LIN {X 0,Y 18.361,Z 633.815,A -85,B 0,C 180,E1 -31180.003,E2 -31180.003} C_VEL
LIN {X 0,Y 12.838,Z 634.499,A -85,B 0,C 180,E1 -31229.96,E2 -31229.96} C_VEL
LIN {X 0,Y 18.335,Z 633.856,A -85,B 0,C 180,E1 -31280.006,E2 -31280.006} C_VEL
LIN {X 0,Y 29.896,Z 631.873,A -85,B 0,C 180,E1 -31300.053,E2 -31300.053} C_VEL
LIN {X 0,Y 43.027,Z 628.501,A -85,B 0,C 180,E1 -31308.471,E2 -31308.471} C_VEL
LIN {X 0,Y 56.614,Z 623.64,A -85,B 0,C 180,E1 -31313.19,E2 -31313.19} C_VEL
LIN {X 0,Y 70.439,Z 617.146,A -85,B 0,C 180,E1 -31316.036,E2 -31316.036} C_VEL
LIN {X 0,Y 82.632,Z 609.917,A -85,B 0,C 180,E1 -31317.76,E2 -31317.76} C_VEL
LIN {X 0,Y 94.884,Z 600.97,A -85,B 0,C 180,E1 -31318.945,E2 -31318.945} C_VEL
LIN {X 0,Y 95.371,Z 600.558,A -85,B 0,C 180,E1 -31318.987,E2 -31318.987} C_VEL
LIN {X 0,Y 98.624,Z 602.092,A -85,B 0,C 180,E1 -31319.255,E2 -31319.255} C_VEL
LIN {X 0,Y 98.624,Z 634.641,A -85,B 0,C 180,E1 -31319.255,E2 -31319.255} C_VEL
LIN {X 0,Y 57.494,Z 634.641,A -85,B 0,C 180,E1 -31319.54,E2 -31319.54} C_VEL
LIN {X 0,Y 55.494,Z 632.641,A -85,B 0,C 180,E1 -31319.565,E2 -31319.565} C_VEL
LIN {X 0,Y 55.494,Z 626.851,A -85,B 0,C 180,E1 -31319.565,E2 -31319.565} C_VEL
LIN {X 0,Y 52.867,Z 624.963,A -85,B 0,C 180,E1 -31319.999,E2 -31319.999} C_VEL
LIN {X 0,Y 42.185,Z 628.5,A -85,B 0,C 180,E1 -31322.018,E2 -31322.018} C_VEL
LIN {X 0,Y 28.271,Z 631.872,A -85,B 0,C 180,E1 -31326.258,E2 -31326.258} C_VEL
LIN {X 0,Y 14.806,Z 633.856,A -85,B 0,C 180,E1 -31338.424,E2 -31338.424} C_VEL
LIN {X 0,Y 5.734,Z 634.499,A -85,B 0,C 180,E1 -31410.089,E2 -31410.089} C_VEL
LIN {X 0,Y 14.912,Z 633.816,A -85,B 0,C 180,E1 -31480.594,E2 -31480.594} C_VEL
LIN {X 0,Y 19.154,Z 633.3,A -85,B 0,C 180,E1 -31486.082,E2 -31486.082} C_VEL
LIN {X 0,Y 20.034,Z 633.15,A -85,B 0,C 180,E1 -31493.272,E2 -31493.272} C_VEL
LIN {X 0,Y 21.231,Z 632.974,A -85,B 0,C 180,E1 -31506.545,E2 -31506.545} C_VEL
LIN {X 0,Y 21.455,Z 632.974,A -85,B 0,C 180,E1 -31510.547,E2 -31510.547} C_VEL
LIN {X 0,Y 8.818,Z 634.324,A -85,B 0,C 180,E1 -31537.063,E2 -31537.063} C_VEL
LIN {X 0,Y 5.734,Z 634.499,A -85,B 0,C 180,E1 -31589.911,E2 -31589.911} C_VEL
LIN {X 0,Y 14.803,Z 633.856,A -85,B 0,C 180,E1 -31661.608,E2 -31661.608} C_VEL
LIN {X 0,Y 28.27,Z 631.872,A -85,B 0,C 180,E1 -31673.77,E2 -31673.77} C_VEL
LIN {X 0,Y 42.184,Z 628.5,A -85,B 0,C 180,E1 -31678.019,E2 -31678.019} C_VEL
LIN {X 0,Y 52.867,Z 624.963,A -85,B 0,C 180,E1 -31679.999,E2 -31679.999} C_VEL
LIN {X 0,Y 52.867,Z 624.963,A -85,B 0,C 180,E1 -31679.999,E2 -31679.999}

QRS_NEXT_CUT()

QRS_NEXT()
QRS_HOME()

END
